{attribute 'GeneratedUsingTerminal: EL9210-0000-0016'}
{attribute addProperty BoxType "EL9210-0000-0016"}
{attribute addProperty Id "FuseErrorAT %I*BOOL1"}
{attribute addProperty CRC "516313306"}
{attribute addProperty Size "1"}
TYPE FuseError_1EC650DA EXTENDS InputBase_8311D824 :
STRUCT
	{attribute addProperty Name "FuseError"}
	FuseError AT %I* : BOOL;
END_STRUCT
END_TYPE

(* stored: Version 1.2.0.0, ProductVersion 3.1.4024.11
   DUT FuseError_1EC650DA: Id {e4ef0648-040e-4b0b-a33e-1724d0df8dcb} *)
